FUNCTION_BLOCK EL3058
VAR
	_io : EL3xx8_Data;
	{attribute addProperty Name "WcState"}
	_wcState : WcStateInputToggle;
	{attribute addProperty Name "Info data"}
	_infoData : InfoDataAds;
END_VAR

PROPERTY IO : REFERENCE TO EL3xx8_Data
GET
IO REF= _io;
END_GET
END_PROPERTY

PROPERTY WcState : REFERENCE TO WcStateInputToggle
GET
WcState REF= _wcState;
END_GET
END_PROPERTY

END_FUNCTION_BLOCK

(* stored: Version 1.1.0.1, ProductVersion 3.1.4024.9
   POU EL3058: Id {36e30ee7-ad42-077c-3c01-f9eb940f65f5}, SpecialFunc None
   Property IO: Id {184d6c99-cfa1-0519-0f14-8048c5b8e9bb}
   Get Get: Id {a3d09683-4332-09dc-05b0-c2a4ec27d28a}
   Property WcState: Id {c89d0e73-c5cb-0648-03d8-2d11eaacc9ba}
   Get Get: Id {d955dae0-81ab-0a72-3b3e-a2ae5d2c7ba1} *)
